// TIA Portal V20 export
VAR_GLOBAL   // PLC tag table "LGR_Const_Task_DragType"
END_VAR
VAR_GLOBAL CONSTANT   // user constants
   DRAGTYPE_1 : Byte := 2#0000_0001;
   DRAGTYPE_2 : Byte := 2#0000_0010;
   DRAGTYPE_3 : Byte := 2#0000_0100;
   DRAGTYPE_4 : Byte := 2#0000_1000;
   DRAGTYPE_5 : Byte := 2#0001_0000;
   DRAGTYPE_6 : Byte := 2#0010_0000;
   DRAGTYPE_7 : Byte := 2#0100_0000;
   DRAGTYPE_8 : Byte := 2#1000_0000;
END_VAR
